// TIA Portal V14 SP1 program export: 0 tag tables, 0 data types, 0 data blocks, 1 code blocks (in call order from the OBs), 0 instance data blocks

ORGANIZATION_BLOCK "Main"   // OB1, LAD, ProgramCycle
TITLE = "Main Program Sweep (Cycle)"
{ S7_Optimized_Access := 'TRUE' }
// stored: CodeModifiedDate 2019-05-02T00:19:22.0356737Z, CompileDate 2019-05-02T00:21:49.3422341Z, CreationDate 2019-05-02T00:12:13.7630248Z, InterfaceModifiedDate 2008-07-21T16:55:08.419547Z, IsConsistent true, ModifiedDate 2019-05-02T00:19:22.0356737Z, ParameterModified 2008-07-21T16:55:08.419547Z, StructureModified 2008-07-21T16:55:08.419547Z
   VAR_INPUT
      Initial_Call : Bool;   // Initial call of this OB
      Remanence : Bool;   // =True, if remanent data are available
   END_VAR
BEGIN

REGION Network 1
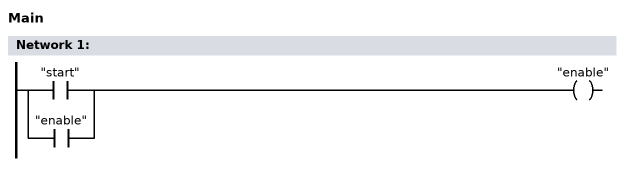
   RUNG wire#powerrail
      Contact( "start" )
      wire#w1
      Coil( "enable" )
   END_RUNG
   RUNG wire#powerrail
      Contact( "enable" )
   END_RUNG wire#w1
   // the same network as SCL:
   "enable" := "start" OR "enable";
END_REGION
END_ORGANIZATION_BLOCK
